(* Schneider Machine Expert - Basic project SHREDDER, file version 2.8.0.0 *)
(* ProjectInformations: Name=Mulino Bazzica *)
(* UserInformations: LastName=Dominici, FirstName=Erica, PhoneNumber=+39 0742 38501, Email=info@promas.com, Street=via XXV Aprile, 10/12, City=Trevi, ZipCode=06039, State=Perugia, Country=Italy *)

HARDWARE
  Cpu 0: TM221CE16T
  EthernetConfiguration: NetworkName=M221, IpAllocationMode=FixedAddress, IpAddress=192.168.0.230, SubnetMask=255.255.254.0
  SerialLineConfiguration: Baud=Baud19200, Parity=ParityEven, DataBits=DataBits8, StopBits=StopBits1, PhysicalMedium=PhysicalMediumRs485, TransmissionMode=TransmissionModeModbusRtu, SlaveId=1, Addressing=SlaveAddressing
  MastTask: UsePeriodScanMode=true, PeriodScan=100
  FastTask: Period=255
  CpuBehavior: StartingMode=StartInRun, AutoSaveRamOnEeprom=true, WatchdogPeriod=250

SYMBOLS  (address, symbol, comment, settings)
  %M0       KM_ALL_ON
  %M1       KM_M1_M2_ON
  %M2       KM_M3_ON
  %MW0      FSM_MILL
  %MW1      M1_M2_OFF_PRESET
  %MW2      M3_OFF_PRESET
  %TM0      TOF_M3  [Type=TOF, Base=OneSecond, IsDynamicPreset=true]
  %TM1      TOF_M1_M2  [Base=OneSecond, IsDynamicPreset=true]
  %TM2      M1_ALM_ON  [Preset=3, Base=OneSecond]
  %TM3      M1_ALM_OFF  [Preset=3, Base=OneSecond]
  %TM4      M2_ALM_ON  [Preset=3, Base=OneSecond]
  %TM5      M2_ALM_OFF  [Preset=3, Base=OneSecond]
  %TM6      M3_ALM_ON  [Preset=3, Base=OneSecond]
  %TM7      M3_ALM_OFF  [Preset=3, Base=OneSecond]
  %I0.0     F1_BOTT_LEV
  %I0.1     F2_UPP_LEV
  %I0.2     START_BTN
  %I0.3     STOP_BTN
  %I0.4     TRIP_OK
  %I0.5     KM1
  %I0.6     KM2
  %I0.7     KM3
  %Q0.0     M1_ON  "MILL"
  %Q0.1     M2_ON  "MILL 2nd MOTOR"
  %Q0.2     M3_ON  "BELT"
  %Q0.3     M1_M2_OFF  "ALL OFF"
  %Q0.4     M3_STOP  "M3 STOP COMMAND"
  %IWM0     FSM_OUT

POU IN
  (* SectionNumber=1 *)

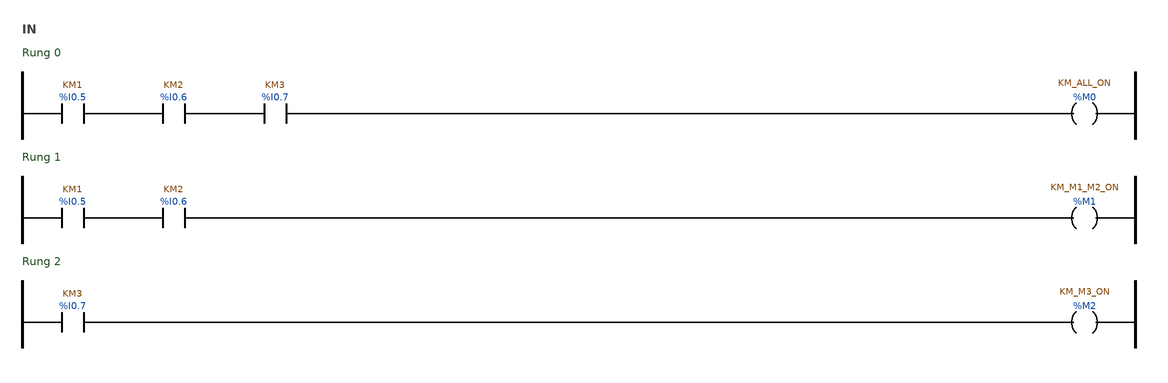

// Rung 0
  LD %I0.5                (* KM1 *)
  AND %I0.6               (* KM2 *)
  AND %I0.7               (* KM3 *)
  ST %M0                  (* KM_ALL_ON *)
  // as ST:
  //   KM_ALL_ON := KM1 AND KM2 AND KM3;

// Rung 1
  LD %I0.5                (* KM1 *)
  AND %I0.6               (* KM2 *)
  ST %M1                  (* KM_M1_M2_ON *)
  // as ST:
  //   KM_M1_M2_ON := KM1 AND KM2;

// Rung 2
  LD %I0.7                (* KM3 *)
  ST %M2                  (* KM_M3_ON *)
  // as ST:
  //   KM_M3_ON := KM3;

POU FSM
  (* SectionNumber=2 *)

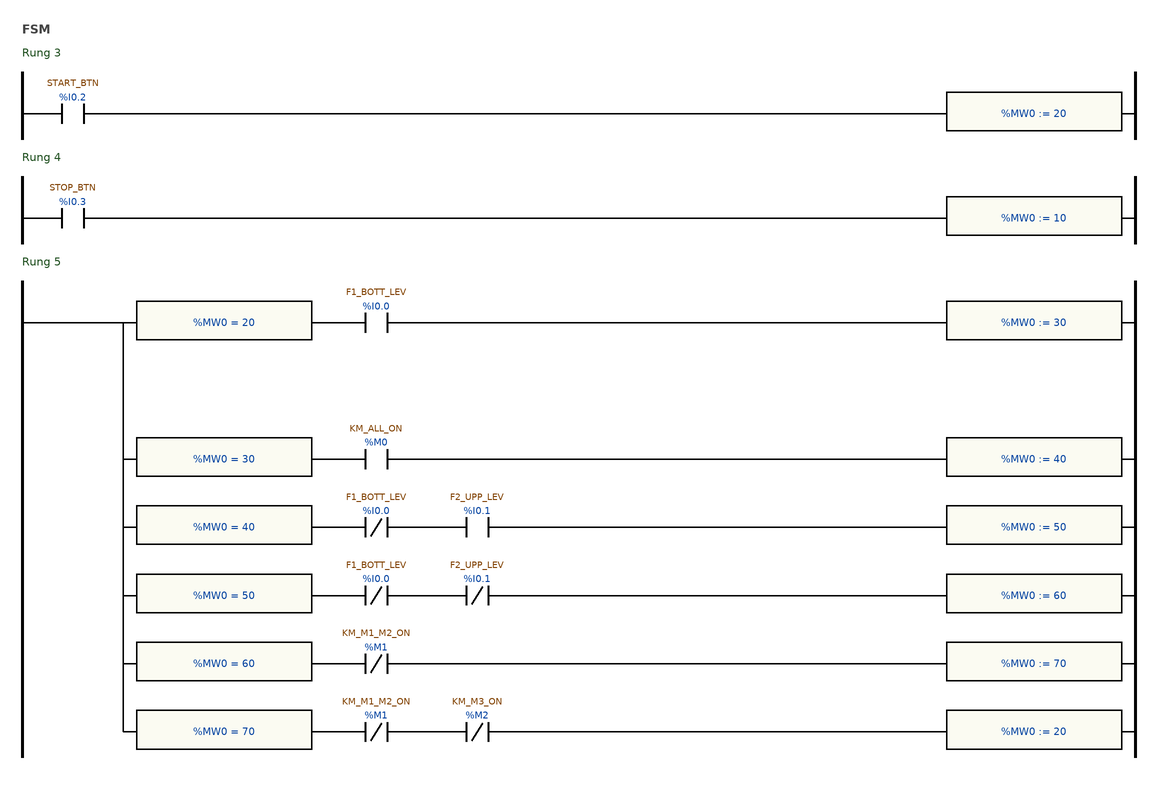

// Rung 3
  LD %I0.2                (* START_BTN *)
  [ %MW0 := 20 ]          (* FSM_MILL *)
  // as ST:
  //   IF START_BTN THEN FSM_MILL := 20; END_IF;

// Rung 4
  LD %I0.3                (* STOP_BTN *)
  [ %MW0 := 10 ]          (* FSM_MILL *)
  // as ST:
  //   IF STOP_BTN THEN FSM_MILL := 10; END_IF;

// Rung 5
  LD 1
  MPS
  AND [ %MW0 = 20 ]       (* FSM_MILL *)
  AND %I0.0               (* F1_BOTT_LEV *)
  [ %MW0 := 30 ]          (* FSM_MILL *)
  MRD
  AND [ %MW0 = 30 ]       (* FSM_MILL *)
  AND %M0                 (* KM_ALL_ON *)
  [ %MW0 := 40 ]          (* FSM_MILL *)
  MRD
  AND [ %MW0 = 40 ]       (* FSM_MILL *)
  ANDN %I0.0              (* F1_BOTT_LEV *)
  AND %I0.1               (* F2_UPP_LEV *)
  [ %MW0 := 50 ]          (* FSM_MILL *)
  MRD
  AND [ %MW0 = 50 ]       (* FSM_MILL *)
  ANDN %I0.0              (* F1_BOTT_LEV *)
  ANDN %I0.1              (* F2_UPP_LEV *)
  [ %MW0 := 60 ]          (* FSM_MILL *)
  MRD
  AND [ %MW0 = 60 ]       (* FSM_MILL *)
  ANDN %M1                (* KM_M1_M2_ON *)
  [ %MW0 := 70 ]          (* FSM_MILL *)
  MPP
  AND [ %MW0 = 70 ]       (* FSM_MILL *)
  ANDN %M1                (* KM_M1_M2_ON *)
  ANDN %M2                (* KM_M3_ON *)
  [ %MW0 := 20 ]          (* FSM_MILL *)
  // as ST:
  //   IF FSM_MILL = 20 AND F1_BOTT_LEV THEN FSM_MILL := 30; END_IF;
  //   IF FSM_MILL = 30 AND KM_ALL_ON THEN FSM_MILL := 40; END_IF;
  //   IF FSM_MILL = 40 AND NOT F1_BOTT_LEV AND F2_UPP_LEV THEN FSM_MILL := 50; END_IF;
  //   IF FSM_MILL = 50 AND NOT F1_BOTT_LEV AND NOT F2_UPP_LEV THEN FSM_MILL := 60; END_IF;
  //   IF FSM_MILL = 60 AND NOT KM_M1_M2_ON THEN FSM_MILL := 70; END_IF;
  //   IF FSM_MILL = 70 AND NOT KM_M1_M2_ON AND NOT KM_M3_ON THEN FSM_MILL := 20; END_IF;

POU TIMERS
  (* SectionNumber=3 *)

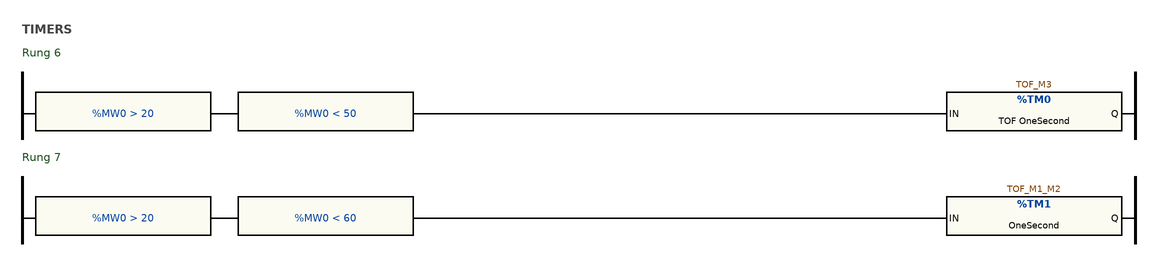

// Rung 6
  BLK %TM0                (* TOF_M3 *)
  LD [ %MW0 > 20 ]        (* FSM_MILL *)
  AND [ %MW0 < 50 ]       (* FSM_MILL *)
  IN
  END_BLK
  // as ST:
  //   TOF_M3(IN := FSM_MILL > 20 AND FSM_MILL < 50);

// Rung 7
  BLK %TM1                (* TOF_M1_M2 *)
  LD [ %MW0 > 20 ]        (* FSM_MILL *)
  AND [ %MW0 < 60 ]       (* FSM_MILL *)
  IN
  END_BLK
  // as ST:
  //   TOF_M1_M2(IN := FSM_MILL > 20 AND FSM_MILL < 60);

POU OUT
  (* SectionNumber=4 *)

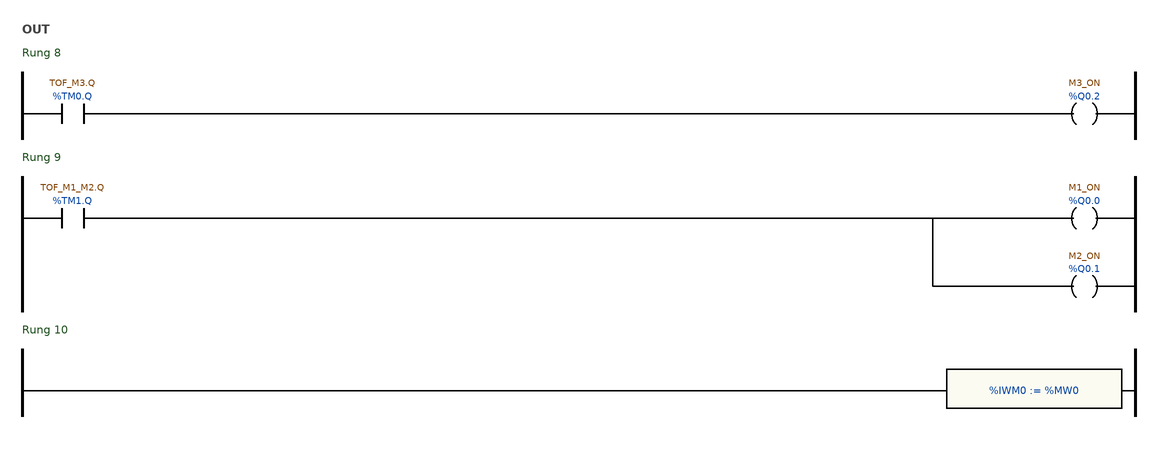

// Rung 8
  LD %TM0.Q               (* TOF_M3 *)
  ST %Q0.2                (* M3_ON *)
  // as ST:
  //   M3_ON := TOF_M3.Q;

// Rung 9
  LD %TM1.Q               (* TOF_M1_M2 *)
  ST %Q0.0                (* M1_ON *)
  ST %Q0.1                (* M2_ON *)
  // as ST:
  //   M1_ON := TOF_M1_M2.Q;
  //   M2_ON := TOF_M1_M2.Q;

// Rung 10
  (* no IL stored for this rung *)

POU SETTINGS
  (* SectionNumber=5 *)

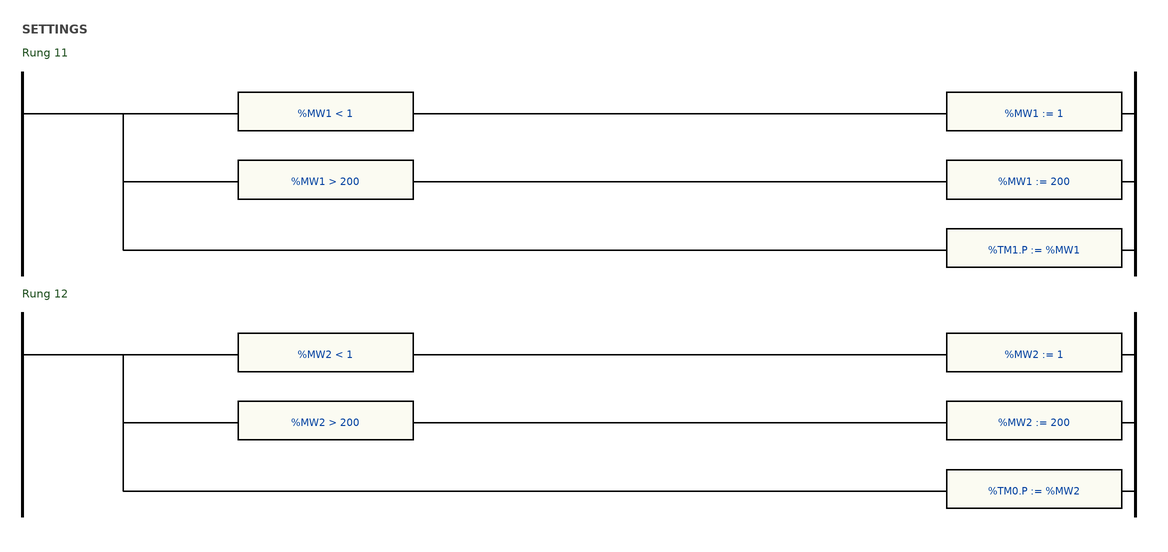

// Rung 11
  LD 1
  MPS
  AND [ %MW1 < 1 ]        (* M1_M2_OFF_PRESET *)
  [ %MW1 := 1 ]           (* M1_M2_OFF_PRESET *)
  MRD
  AND [ %MW1 > 200 ]      (* M1_M2_OFF_PRESET *)
  [ %MW1 := 200 ]         (* M1_M2_OFF_PRESET *)
  MPP
  [ %TM1.P := %MW1 ]      (* TOF_M1_M2, M1_M2_OFF_PRESET *)
  // as ST:
  //   IF M1_M2_OFF_PRESET < 1 THEN M1_M2_OFF_PRESET := 1; END_IF;
  //   IF M1_M2_OFF_PRESET > 200 THEN M1_M2_OFF_PRESET := 200; END_IF;
  //   TOF_M1_M2.P := M1_M2_OFF_PRESET;

// Rung 12
  LD 1
  MPS
  AND [ %MW2 < 1 ]        (* M3_OFF_PRESET *)
  [ %MW2 := 1 ]           (* M3_OFF_PRESET *)
  MRD
  AND [ %MW2 > 200 ]      (* M3_OFF_PRESET *)
  [ %MW2 := 200 ]         (* M3_OFF_PRESET *)
  MPP
  [ %TM0.P := %MW2 ]      (* TOF_M3, M3_OFF_PRESET *)
  // as ST:
  //   IF M3_OFF_PRESET < 1 THEN M3_OFF_PRESET := 1; END_IF;
  //   IF M3_OFF_PRESET > 200 THEN M3_OFF_PRESET := 200; END_IF;
  //   TOF_M3.P := M3_OFF_PRESET;

POU ALARMS
  (* SectionNumber=6 *)

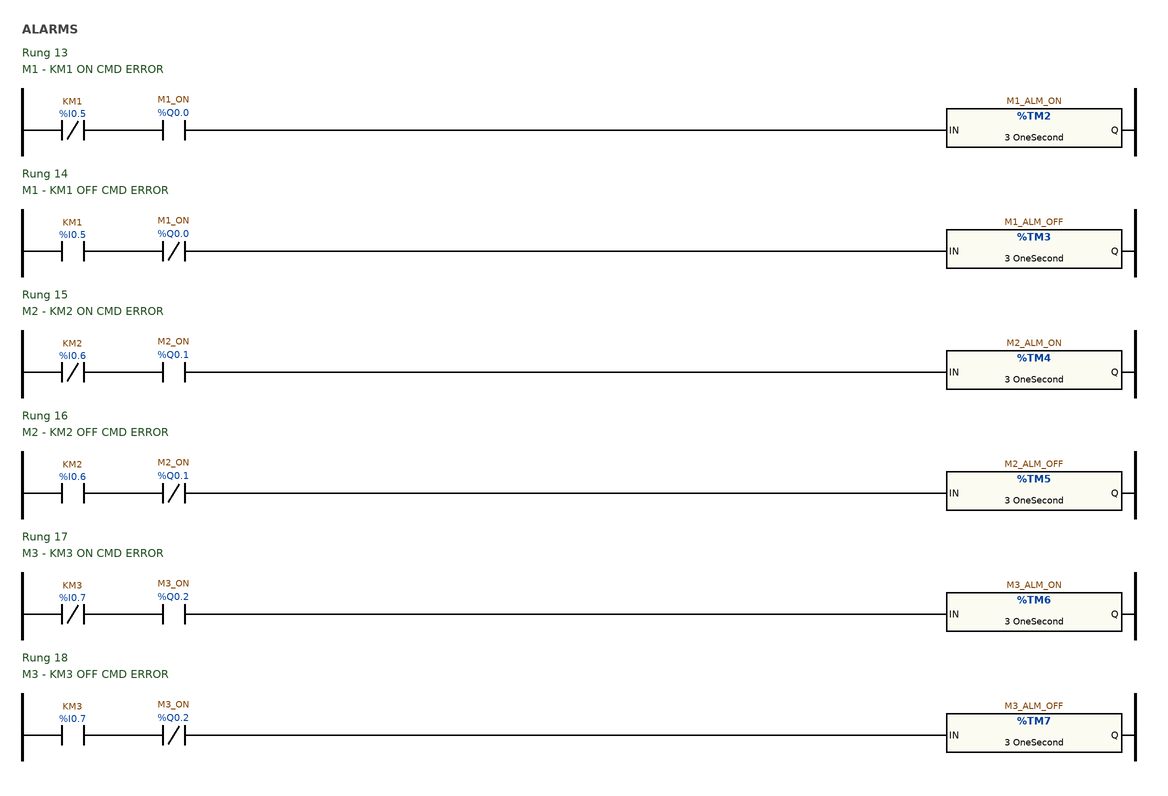

// Rung 13
// M1 - KM1 ON CMD ERROR
  BLK %TM2                (* M1_ALM_ON *)
  LDN %I0.5               (* KM1 *)
  AND %Q0.0               (* M1_ON *)
  IN
  END_BLK
  // as ST:
  //   M1_ALM_ON(IN := NOT KM1 AND M1_ON);

// Rung 14
// M1 - KM1 OFF CMD ERROR
  BLK %TM3                (* M1_ALM_OFF *)
  LD %I0.5                (* KM1 *)
  ANDN %Q0.0              (* M1_ON *)
  IN
  END_BLK
  // as ST:
  //   M1_ALM_OFF(IN := KM1 AND NOT M1_ON);

// Rung 15
// M2 - KM2 ON CMD ERROR
  BLK %TM4                (* M2_ALM_ON *)
  LDN %I0.6               (* KM2 *)
  AND %Q0.1               (* M2_ON *)
  IN
  END_BLK
  // as ST:
  //   M2_ALM_ON(IN := NOT KM2 AND M2_ON);

// Rung 16
// M2 - KM2 OFF CMD ERROR
  BLK %TM5                (* M2_ALM_OFF *)
  LD %I0.6                (* KM2 *)
  ANDN %Q0.1              (* M2_ON *)
  IN
  END_BLK
  // as ST:
  //   M2_ALM_OFF(IN := KM2 AND NOT M2_ON);

// Rung 17
// M3 - KM3 ON CMD ERROR
  BLK %TM6                (* M3_ALM_ON *)
  LDN %I0.7               (* KM3 *)
  AND %Q0.2               (* M3_ON *)
  IN
  END_BLK
  // as ST:
  //   M3_ALM_ON(IN := NOT KM3 AND M3_ON);

// Rung 18
// M3 - KM3 OFF CMD ERROR
  BLK %TM7                (* M3_ALM_OFF *)
  LD %I0.7                (* KM3 *)
  ANDN %Q0.2              (* M3_ON *)
  IN
  END_BLK
  // as ST:
  //   M3_ALM_OFF(IN := KM3 AND NOT M3_ON);
